// TIA Portal V21 export
// export: Created 2026-08-11T14:59:46Z, ExportSetting WithDefaults
VAR_GLOBAL   // PLC tag table "Inputs"
   EStop_Ok AT %I0.0 : Bool;   // E-stop status contact - E-stop status contact (NC, TRUE = released)
   GuardDoor_Ok AT %I0.1 : Bool;   // Transfer guard door switch - guard status contact (NC, TRUE = closed)
   StartPb AT %I0.2 : Bool;   // Cycle start pushbutton
   StopPb AT %I0.3 : Bool;   // Cycle stop pushbutton
   ResetPb AT %I0.4 : Bool;   // Fault reset pushbutton
   PartPresent AT %I0.5 : Bool;   // Part present at infeed
   PartAtOutfeed AT %I0.6 : Bool;   // Part arrived at outfeed
   Infeed_Running AT %I0.7 : Bool;   // Infeed conveyor - aux contact
   Infeed_Fault AT %I1.0 : Bool;   // Infeed conveyor - overload contact
   Clamp_Opened AT %I1.1 : Bool;   // Part clamp - open limit switch
   Clamp_Closed AT %I1.2 : Bool;   // Part clamp - closed limit switch
   Lift_Opened AT %I1.3 : Bool;   // Transfer lift - open limit switch
   Lift_Closed AT %I1.4 : Bool;   // Transfer lift - closed limit switch
   Outfeed_Running AT %I1.5 : Bool;   // Outfeed conveyor drive - drive running
   Outfeed_Fault AT %I1.6 : Bool;   // Outfeed conveyor drive - drive fault
END_VAR
